INTERFACE I_AsynchronousRpcResponseFactory

METHOD PUBLIC Create : I_AsynchronousRpcResponse
VAR_INPUT
END_VAR
END_METHOD

END_INTERFACE

(* stored: Version 1.1.0.1, ProductVersion 3.1.4024.12
   Itf I_AsynchronousRpcResponseFactory: Id {6d5e561e-cbcb-4c30-b95b-e726f88dfa68}
   Method Create: Id {27c8f483-4ceb-4c4a-aa95-0abeffe3f05a} *)
